INTERFACE I_CommsTransceiver EXTENDS I_CommsReceiver, I_CommsTransmitter

END_INTERFACE

(* stored: Version 1.1.0.1, ProductVersion 3.1.4024.9
   Itf I_CommsTransceiver: Id {92621764-4666-437c-b4b6-8f4edc88ce6c} *)
